// TIA Portal V18 export
VAR_GLOBAL   // PLC tag table "02  Costanti SAFETY_DEVICE"
END_VAR
VAR_GLOBAL CONSTANT   // user constants
   SBF : DInt := 1;   // Fungo emergenza
   SBAA : DInt := 2;   // Abilita potenza
   BF1 : DInt := 3;   // Barriere fotoelettriche monoraggio
   BFM : DInt := 4;   // Barriere fotoelettriche multiraggio
   TCR : DInt := 5;   // Cancelli e ripari gestiti con transponder
   Z1 : Int := 1;
   Z2 : Int := 2;
   Z3 : Int := 3;
   Z4 : Int := 4;
   Z5 : Int := 5;
   SCE : DInt := 5;   // Elettroserratura
   SBAN : DInt := 5;   // Banderuola sicurezza
   "BY-PASS" : DInt := 6;   // Chiave di by pass inserita
END_VAR
